// TIA Portal V17 export
// export: Created 2024-12-18T10:10:48.3541596Z, ExportSetting WithDefaults, DisplayName Totally Integrated Automation Portal, DisplayVersion V17, DisplayName TIA Portal Openness, DisplayVersion V17, DisplayName TIA Portal Version Control Interface, DisplayVersion V17, DisplayName STEP 7 Professional, DisplayVersion V17, DisplayName STEP 7 Safety, DisplayVersion V17, DisplayName WinCC Advanced / Unified PC, DisplayVersion V17
FUNCTION_BLOCK "Last version"   // FB6, LAD
{ S7_Optimized_Access := 'TRUE' }
VERSION : 0.1
// stored: AutoNumber true, IsIECCheckEnabled false, IsRetainMemResEnabled false, MemoryReserve 100, SetENOAutomatically false, UDAEnableTagReadback false
BEGIN

REGION Network 2: Calculate Flow
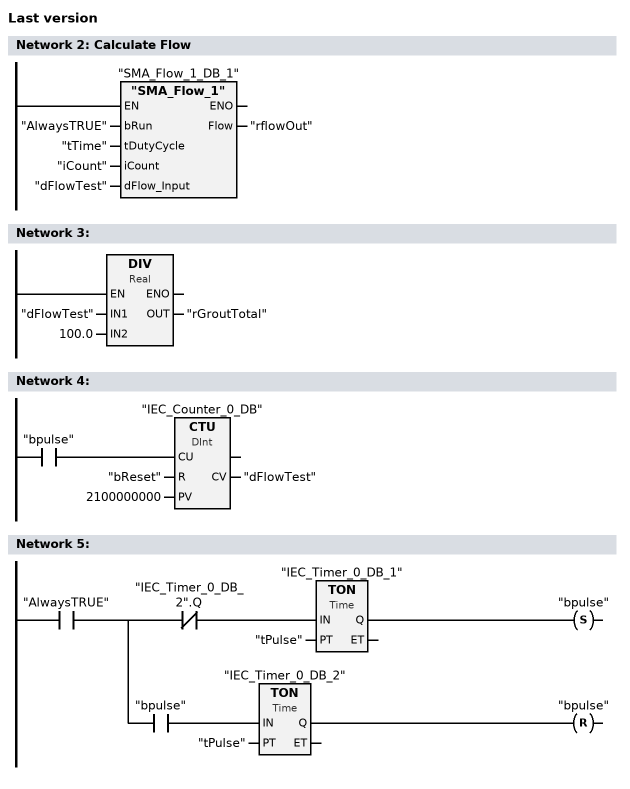
   RUNG wire#powerrail
      "SMA_Flow_1_DB_1"(bRun := "AlwaysTRUE", tDutyCycle := "tTime", iCount := "iCount", dFlow_Input := "dFlowTest", Flow => "rflowOut")
   END_RUNG
   // the same network as SCL:
   "SMA_Flow_1_DB_1"(bRun := "AlwaysTRUE",   // "SMA_Flow_1"
                     tDutyCycle := "tTime",
                     iCount := "iCount",
                     dFlow_Input := "dFlowTest",
                     Flow => "rflowOut");
END_REGION

REGION Network 3
   RUNG wire#powerrail
      { S7_Templates := "SrcType := Real" } Div(in1 := "dFlowTest", in2 := 100.0, out => "rGroutTotal")
   END_RUNG
   // the same network as SCL:
   "rGroutTotal" := "dFlowTest" / 100.0;
END_REGION

REGION Network 4
   RUNG wire#powerrail
      Contact( "bpulse" )
      { S7_Templates := "value_type := DInt" } "IEC_Counter_0_DB".CTU(r := "bReset", pv := 2100000000, cv => "dFlowTest")
   END_RUNG
   // the same network as SCL:
   "IEC_Counter_0_DB".CTU(CU := "bpulse", R := "bReset", PV := 2100000000, CV => "dFlowTest");
END_REGION

REGION Network 5
   RUNG wire#powerrail
      Contact( "AlwaysTRUE" )
      wire#w1
      I_Contact( "IEC_Timer_0_DB_2".Q )
      { S7_Templates := "time_type := Time" } "IEC_Timer_0_DB_1".TON(pt := "tPulse", et =>)
      S_Coil( "bpulse" )
   END_RUNG
   RUNG wire#w1
      Contact( "bpulse" )
      { S7_Templates := "time_type := Time" } "IEC_Timer_0_DB_2".TON(pt := "tPulse", et =>)
      R_Coil( "bpulse" )
   END_RUNG
   // the same network as SCL:
   "IEC_Timer_0_DB_1".TON(IN := "AlwaysTRUE" AND NOT "IEC_Timer_0_DB_2".Q, PT := "tPulse");
   IF "IEC_Timer_0_DB_1".Q THEN "bpulse" := TRUE; END_IF;
   "IEC_Timer_0_DB_2".TON(IN := "AlwaysTRUE" AND "bpulse", PT := "tPulse");
   IF "IEC_Timer_0_DB_2".Q THEN "bpulse" := FALSE; END_IF;
END_REGION

REGION Network 6: Start ReCording...
END_REGION
END_FUNCTION_BLOCK
